# B&R Automation Studio project Server
Automation Studio 6.5.2.12; technology packages: mappCockpit 6.6.0, mappConnect 6.1.0, mappServices 6.6.0, mappView 6.6.0, OpcUaCs 6.6.1

## Configuration Demo

CPU PC_any, AutomationRuntime 6.6.2, Build 11.3.0, Vc 6.5.0

### Task classes (Cpu.sw)
```
Cyclic#1 (cycle 10000 us):
  Program <- Program.prg
Libraries: standard, runtime, AsZip, FileIO, CoTrace
```

### Hardware
```
PC : PC_any v1.1.2.0 (OrderNumber=PC)
  ConfigurationID = Server_Demo
  Cyclic1Duration = 10000
  FileDevice1
  FileDeviceName1 = USER
  FileDevicePath1 = USER_PATH
```

### BRRole.brrole - PC/AccessAndSecurity/UserRoleSystem/BRRole.brrole
```
Element BR_Anonymous (Type=BRRole)
Element BR_Engineer (Type=BRRole)
Element BR_Observer (Type=BRRole)
Element BR_SafetyAdmin (Type=BRRole)
Element BR_SecurityAdmin (Type=BRRole)
```

- Physical/Demo/PC/IoMap.iom: same as Physical/Demo/PC/Cpu.per
- Physical/Demo/PC/PvMap.vvm: same as Physical/Demo/PC/Cpu.per
### Config.mappconnect - PC/mappConnect/Config.mappconnect
```
Element mapp Connect Configuration (Type=mappconnect)
  WebServerProtocol:
    WebServerPortSsl = 8443
    Interface = All
    SSLConfiguration
  WebServerEndpointConfiguration:
    Endpoint[1]:
      Endpoint = /*
      Roles:
        Role[1] = BR_Anonymous
        Role[2] = BR_Engineer
  OpcUaServerWhitelist:
    OpcUaServer[1]:
      Url = opc.tcp://127.0.0.1:4840
```

- Safety project (password-protected, skipped)

## Logical view

Binary libraries used (declarations not repeated): operator, runtime, AsIecCon, standard, AsZip, FileIO, CoTrace 6.6.0

### Global.typ - Global data types
```iecst
(*
     * HMIDemo types
     *
     * Shared state between the HMIDemo PLC task and the lux-react demo HMI.
     * All fields are accessible as OPC UA nodes under the variable name 'HMIDemo'.
     *
     * Example OPC UA paths:
     *   HMIDemo.Power                  — written by HMI
     *   HMIDemo.Speed                  — read by HMI
     *   HMIDemo.Settings.SpeedLimit    — read/write
     *   HMIDemo.Recipes.Slots[0].Name  — read
     *   HMIDemo.Alarms.TempHigh        — read
     *)

TYPE
	HMIDemo_Settings_typ : STRUCT
		SpeedLimit : REAL; (* Maximum allowed speed (RPM)       *)
		TempWarnThreshold : REAL; (* Temperature warning level (°C)    *)
		PressureWarnThreshold : REAL; (* Pressure warning level (bar)      *)
		AutoStopOnAlarm : BOOL; (* Auto-stop motor when alarm active *)
	END_STRUCT;

	HMIDemo_Recipe_typ : STRUCT
		Name : STRING[40]; (* Recipe display name               *)
		Setpoint : REAL; (* Speed setpoint (RPM)              *)
		PressureTarget : REAL; (* Target pressure (bar)             *)
	END_STRUCT;

	HMIDemo_Recipes_typ : STRUCT
		ActiveIndex : USINT; (* Recipe index to load (0..3)       *)
		Load : BOOL; (* HMI sets TRUE to load recipe      *)
		LoadedIndex : USINT; (* Currently loaded recipe index     *)
		Slots : ARRAY[0..3] OF HMIDemo_Recipe_typ;
	END_STRUCT;

	HMIDemo_Alarms_typ : STRUCT
		TempHigh : BOOL; (* Temperature above threshold       *)
		PressureHigh : BOOL; (* Pressure above threshold          *)
		SpeedFault : BOOL; (* Speed exceeds limit               *)
		AnyActive : BOOL; (* OR of all alarm conditions        *)
		AckAll : BOOL; (* HMI sets TRUE to acknowledge      *)
	END_STRUCT;

	HMIDemo_typ : STRUCT
		(* ---- Commands (HMI -> PLC) ---- *)
		Power : BOOL; (* TRUE = run, FALSE = stop          *)
		Setpoint : REAL; (* Speed setpoint (RPM)              *)
		PressureTarget : REAL; (* Pressure target (bar)             *)
		(* ---- Status  (PLC -> HMI) ---- *)
		Speed : REAL; (* Actual motor speed (RPM)          *)
		Temp : REAL; (* Motor temperature (°C)            *)
		Running : BOOL; (* Motor is running                  *)
		Pressure : REAL; (* Hydraulic pressure (bar)          *)
		Status : STRING[80]; (* Status text                       *)
		Heartbeat : BOOL; (* Toggled by PLC every 500 ms       *)
		Cycles : UDINT; (* Cycle counter                     *)
		(* ---- Sub-structures ---- *)
		Settings : HMIDemo_Settings_typ;
		Recipes : HMIDemo_Recipes_typ;
		Alarms : HMIDemo_Alarms_typ;
	END_STRUCT;
END_TYPE
```

### Global.var
```iecst
VAR
    HMIDemo : HMIDemo_typ;
END_VAR
```


### Program Logical/Program (IEC)

#### Cyclic.st - Cyclic code
```iecst
PROGRAM _CYCLIC

(* ------------------------------------------------------------------ *)
(*  HMIDemoTask  CYCLIC                                               *)
(*  Default task class: #Cyclic, recommended cycle time: 100ms.       *)
(* ------------------------------------------------------------------ *)

(* 1. Heartbeat  toggle every 500 ms -------------------------------- *)
	tHeartbeat(IN := NOT tHeartbeat.Q, PT := T#500ms);
	IF tHeartbeat.Q THEN
		HMIDemo.Heartbeat := NOT HMIDemo.Heartbeat;
	END_IF

(* 2. Clamp setpoint to speed limit --------------------------------- *)
	IF HMIDemo.Setpoint > HMIDemo.Settings.SpeedLimit THEN
		HMIDemo.Setpoint := HMIDemo.Settings.SpeedLimit;
	END_IF

(* 3. Motor speed  ramp toward setpoint when powered,
      ramp to zero when stopped -------------------------------------- *)
	IF HMIDemo.Power THEN
		IF HMIDemo.Speed < HMIDemo.Setpoint THEN
			HMIDemo.Speed := MIN(HMIDemo.Speed + 50.0, HMIDemo.Setpoint);
		ELSIF HMIDemo.Speed > HMIDemo.Setpoint THEN
			HMIDemo.Speed := MAX(HMIDemo.Speed - 50.0, HMIDemo.Setpoint);
		END_IF
	ELSE
		HMIDemo.Speed := MAX(HMIDemo.Speed - 80.0, 0.0);
	END_IF

	HMIDemo.Running := HMIDemo.Speed > 10.0;

(* 4. Motor temperature  22 + (speed * 0.06) ------------------------ *)
	HMIDemo.Temp := 22.0 + (HMIDemo.Speed * 0.06);

(* 5. Hydraulic pressure  builds toward target when running ---------- *)
	IF HMIDemo.Running THEN
		HMIDemo.Pressure := MIN(HMIDemo.Pressure + 10.0, HMIDemo.PressureTarget);
	ELSE
		HMIDemo.Pressure := MAX(HMIDemo.Pressure - 5.0, 0.0);
	END_IF

(* 6. Cycle counter  increment every 2 s while running --------------- *)
	tCycle(IN := HMIDemo.Running AND NOT tCycle.Q, PT := T#2s);
	IF tCycle.Q THEN
		HMIDemo.Cycles := HMIDemo.Cycles + 1;
	END_IF

(* 7. Status text ---------------------------------------------------- *)
	IF HMIDemo.Running THEN
		HMIDemo.Status := 'RUNNING';
	ELSIF HMIDemo.Speed > 0.0 THEN
		HMIDemo.Status := 'STOPPING';
	ELSIF HMIDemo.Power THEN
		HMIDemo.Status := 'STARTING';
	ELSE
		HMIDemo.Status := 'IDLE';
	END_IF

(* 8. Recipe loading ------------------------------------------------- *)
	IF HMIDemo.Recipes.Load THEN
		HMIDemo.Setpoint       := HMIDemo.Recipes.Slots[HMIDemo.Recipes.ActiveIndex].Setpoint;
		HMIDemo.PressureTarget := HMIDemo.Recipes.Slots[HMIDemo.Recipes.ActiveIndex].PressureTarget;
		HMIDemo.Recipes.LoadedIndex := HMIDemo.Recipes.ActiveIndex;
		HMIDemo.Recipes.Load   := FALSE;
	END_IF

(* 9. Alarm evaluation ----------------------------------------------- *)
	HMIDemo.Alarms.TempHigh     := HMIDemo.Temp     > HMIDemo.Settings.TempWarnThreshold;
	HMIDemo.Alarms.PressureHigh := HMIDemo.Pressure  > HMIDemo.Settings.PressureWarnThreshold;
	HMIDemo.Alarms.SpeedFault   := HMIDemo.Speed     > HMIDemo.Settings.SpeedLimit;
	HMIDemo.Alarms.AnyActive    := HMIDemo.Alarms.TempHigh
	                             OR HMIDemo.Alarms.PressureHigh
	                             OR HMIDemo.Alarms.SpeedFault;

(* 10. Auto-stop on alarm -------------------------------------------- *)
	IF HMIDemo.Settings.AutoStopOnAlarm AND HMIDemo.Alarms.AnyActive THEN
		HMIDemo.Power := FALSE;
	END_IF

(* 11. Acknowledge reset --------------------------------------------- *)
	IF HMIDemo.Alarms.AckAll THEN
		HMIDemo.Alarms.AckAll := FALSE;
	END_IF

END_PROGRAM
```

#### Init.st - Init code
```iecst
PROGRAM _INIT
	(* ---- Motor / system defaults ---- *)
	HMIDemo.Status         := 'IDLE';
	HMIDemo.Speed          := 0.0;
	HMIDemo.Temp           := 22.0;
	HMIDemo.Pressure       := 0.0;
	HMIDemo.PressureTarget := 180.0;
	HMIDemo.Running        := FALSE;
	HMIDemo.Heartbeat      := FALSE;
	HMIDemo.Cycles         := 0;

	(* ---- Settings defaults ---- *)
	HMIDemo.Settings.SpeedLimit             := 2500.0;
	HMIDemo.Settings.TempWarnThreshold      := 60.0;
	HMIDemo.Settings.PressureWarnThreshold  := 160.0;
	HMIDemo.Settings.AutoStopOnAlarm        := FALSE;

	(* ---- Recipe presets ---- *)
	HMIDemo.Recipes.LoadedIndex := 0;

	HMIDemo.Recipes.Slots[0].Name           := 'Slow';
	HMIDemo.Recipes.Slots[0].Setpoint       := 500.0;
	HMIDemo.Recipes.Slots[0].PressureTarget := 80.0;

	HMIDemo.Recipes.Slots[1].Name           := 'Medium';
	HMIDemo.Recipes.Slots[1].Setpoint       := 1500.0;
	HMIDemo.Recipes.Slots[1].PressureTarget := 120.0;

	HMIDemo.Recipes.Slots[2].Name           := 'Fast';
	HMIDemo.Recipes.Slots[2].Setpoint       := 2500.0;
	HMIDemo.Recipes.Slots[2].PressureTarget := 160.0;

	HMIDemo.Recipes.Slots[3].Name           := 'Custom';
	HMIDemo.Recipes.Slots[3].Setpoint       := 0.0;
	HMIDemo.Recipes.Slots[3].PressureTarget := 0.0;
END_PROGRAM
```

#### Exit.st - Exit code
```iecst
PROGRAM _EXIT
	(* Insert code here *)

END_PROGRAM
```

#### Variables.var - Local variables
```iecst
VAR
	tHeartbeat : TON;   (* 500 ms heartbeat toggle timer *)
	tCycle     : TON;   (* 2-second cycle counter timer  *)
END_VAR

VAR CONSTANT

END_VAR
```
